// TwinCAT 3 PLC project Times
// Title: Times
// Company: TomasRompotl
// ProjectVersion: 0.0.1
// ProgramVersion: 3.1.4024.0
// libraries:
//   MachineBase, * (TomasRompotl)
//   Strings, * (TomasRompotl)
//   Tc2_Standard, * (Beckhoff Automation GmbH)
//   Tc2_System, * (Beckhoff Automation GmbH)
//   Tc2_Utilities, * (Beckhoff Automation GmbH)
// project tree:
//   Clocks/ PeriodicTrigger.TcPOU (not stored)
//   Convert/ SecondsToTime.TcPOU, TimeToSeconds.TcPOU
//   CycleTime/ GetCycleTimeInSeconds.TcPOU (not stored)
//   TimeProvider/ TimeProvider.TcPOU (not stored)
//   Version/ Global_Version.TcGVL
// (motion and I/O tree: see PLC project types)
// real-time tasks:
//   TASK BindingTestTask: cycle T#10ms, priority 20, ADS port 350
//   TASK PlcTask: cycle T#10ms, priority 21, ADS port 351
//   TASK PlcTask1: cycle T#10ms, priority 22, ADS port 352
//   TASK PlcTask2: cycle T#10ms, priority 23, ADS port 353

// ---- Version/Global_Version.TcGVL
{attribute 'TcGenerated'}
{attribute 'no-analysis'}
{attribute 'linkalways'}
// This function has been automatically generated from the project information.
VAR_GLOBAL CONSTANT
	{attribute 'const_non_replaced'}
	stLibVersion_Times : ST_LibVersion := (iMajor := 0, iMinor := 0, iBuild := 1, iRevision := 0, nFlags := 0, sVersion := '0.0.1');
END_VAR

// ---- Convert/SecondsToTime.TcPOU
FUNCTION SecondsToTime : TIME
VAR_INPUT
	seconds : LREAL;
END_VAR

SecondsToTime := LREAL_TO_TIME(seconds * 1000);

END_FUNCTION

// ---- Convert/TimeToSeconds.TcPOU
FUNCTION TimeToSeconds : LREAL
VAR_INPUT
	t : TIME;
END_VAR

TimeToSeconds := TIME_TO_LREAL(t) * 0.001;

END_FUNCTION
